FUNCTION_BLOCK FB_MotorTestSuite EXTENDS TcUnit.FB_TestSuite
(*
    Base class for motion tests.

    Contains some helper methods that would otherwise need to be instantiated many times,
    but in this form can be accessed quickly and succinctly in the test suite.
*)

METHOD SetEnables
(*
    Set a motion stage's enables such that it is fully allowed to move.
*)
VAR_IN_OUT
    stMotionStage: ST_MotionStage;
END_VAR
stMotionStage.bHardwareEnable := TRUE;
stMotionStage.bLimitBackwardEnable := TRUE;
stMotionStage.bLimitForwardEnable := TRUE;
stMotionStage.bPowerSelf := TRUE;
END_METHOD

METHOD SetEnablesPMPS
(*
    Set a motion stage's enables such that only PMPS would be preventing a move.
*)
VAR_IN_OUT
    stMotionStage: ST_MotionStage;
END_VAR

SetEnables(stMotionStage);
stMotionStage.bPowerSelf := FALSE;
END_METHOD

METHOD SetGoodState
(*
    Mark a state as valid and ready to use.
*)
VAR_IN_OUT
    stPositionState: ST_PositionState;
END_VAR
stPositionState.bMoveOk := TRUE;
stPositionState.bValid := TRUE;
END_METHOD

END_FUNCTION_BLOCK

(* stored: Version 1.1.0.1
   POU FB_MotorTestSuite: Id {62209a82-679e-47f8-9b5a-ad180dcad4e7}, SpecialFunc None
   Method SetEnables: Id {9a689027-7edb-4bec-9a75-8e1dc053d941}
   Method SetEnablesPMPS: Id {29072525-240d-4c4a-8b5e-95863d0109d6}
   Method SetGoodState: Id {b3c6256b-7995-4ca9-aaf3-c136e49e66c8} *)
